// TIA Portal V15.1 export
// export: Created 2024-06-21T08:40:59.2288324Z, ExportSetting WithDefaults, DisplayName Totally Integrated Automation Portal, DisplayVersion V15.1 Update 5, DisplayName TIA Portal Openness, DisplayVersion V15.1 Update 5, DisplayName SINAMICS Startdrive Advanced, DisplayVersion V15.1, DisplayName G130, G150, S120, S150, SINAMICS MV, S210, DisplayVersion V15.1, DisplayName G110M, G120, G120C, G120D, G120P, DisplayVersion V15.1, DisplayName STEP 7 Professional, DisplayVersion V15.1 Update 5, DisplayName STEP 7 Safety, DisplayVersion V15.1, DisplayName WinCC Professional, DisplayVersion V15.1 Update 5, DisplayName SIMATIC Visualization Architect, DisplayVersion V15.1
FUNCTION_BLOCK "LVDComSubSystemS7-1500"   // FB2215, FBD
TITLE = VDComSubSystemS7-1500
{ S7_Optimized_Access := 'FALSE' }
AUTHOR : VCC
FAMILY : Communic
VERSION : 0.1
// =============================================================================
// This Module Extract Data From VDCom Send/Recv
// =============================================================================
// stored: AutoNumber false, IsIECCheckEnabled false, SetENOAutomatically False, UDAEnableTagReadback false
   VAR_INPUT
      I_CommunicationReset { ExternalAccessible := 'False'; ExternalVisible := 'False'; ExternalWritable := 'False'} : Bool;   // Reset communication by Application
      I_SendRequest { ExternalAccessible := 'False'; ExternalVisible := 'False'; ExternalWritable := 'False'} : Bool;   // Send Command by Application
      I_ResetNewData { ExternalAccessible := 'False'; ExternalVisible := 'False'; ExternalWritable := 'False'} : Bool;   // Trigger by Application to Reset output "NewData"
      I_MasterNewMessage { ExternalAccessible := 'False'; ExternalVisible := 'False'; ExternalWritable := 'False'} : Bool;   // Signal from MasterBlock to indicate new message.
      I_MasterSendFinished { ExternalAccessible := 'False'; ExternalVisible := 'False'; ExternalWritable := 'False'} : Bool;   // Acknowledge from MasterBlock that Send command has been performed
      I_VDCommRecvDB { ExternalAccessible := 'False'; ExternalVisible := 'False'; ExternalWritable := 'False'} : DB_ANY;   // VD communication system receive DB; Not to be used by Application
      I_VDCommSendDB { ExternalAccessible := 'False'; ExternalVisible := 'False'; ExternalWritable := 'False'} : DB_ANY;   // VD communication system send DB; Not to be used by Application
      C_LocalRecvDB { ExternalAccessible := 'False'; ExternalVisible := 'False'; ExternalWritable := 'False'} : DB_ANY;   // Local DB For Recv Data Used By The Application
      C_LocalSendDB { ExternalAccessible := 'False'; ExternalVisible := 'False'; ExternalWritable := 'False'} : DB_ANY;   // Local DB For Send Data Used By The Application
      C_MessType { ExternalAccessible := 'False'; ExternalVisible := 'False'; ExternalWritable := 'False'} : Int := 10;   // Identify Message
      C_SubSystem { ExternalAccessible := 'False'; ExternalVisible := 'False'; ExternalWritable := 'False'} : Int;   // Identify Subsystem
      C_SendMessLen { ExternalAccessible := 'False'; ExternalVisible := 'False'; ExternalWritable := 'False'} : Word;   // Number to identify the Length of the message
   END_VAR
   VAR_OUTPUT
      O_SendFinished { ExternalAccessible := 'False'; ExternalVisible := 'False'; ExternalWritable := 'False'} : Bool;   // Sending of Data is done; to Application
      O_NewData { ExternalAccessible := 'False'; ExternalVisible := 'False'; ExternalWritable := 'False'} : Bool;   // New data is available from SubSystem to Application
   END_VAR
   VAR_IN_OUT
      IO_MasterSendReq { ExternalAccessible := 'False'; ExternalVisible := 'False'; ExternalWritable := 'False'} : Bool;   // Request from the SubBlock to the MasterBlock to Send data
      IO_MasterAckReq { ExternalAccessible := 'False'; ExternalVisible := 'False'; ExternalWritable := 'False'} : Bool;   // Acknowledge to Master upon MessageType- and SubSystem Match
      IO_SubSystemDBNr { ExternalAccessible := 'False'; ExternalVisible := 'False'; ExternalWritable := 'False'} : Int;   // VD Communication Send DB number, Set by SubSystem
      IO_VDCommSendDB { ExternalAccessible := 'False'; ExternalVisible := 'False'; ExternalWritable := 'False'} : DB_ANY;   // VD Communication send DB
   END_VAR
   VAR DB_SPECIFIC
      ThisModuleActiveSend { ExternalAccessible := 'False'; ExternalVisible := 'False'; ExternalWritable := 'False'} : Bool;   // This module active for sending
      ThisModuleActiveRead { ExternalAccessible := 'False'; ExternalVisible := 'False'; ExternalWritable := 'False'} : Bool;   // This module active for Reading / acknowledge
      NewDataPulse { ExternalAccessible := 'False'; ExternalVisible := 'False'; ExternalWritable := 'False'} : Bool;   // Bit to create pulse on NewData
      NewData { ExternalAccessible := 'False'; ExternalVisible := 'False'; ExternalWritable := 'False'} : Bool;   // New Data
      NewDataAvailable { ExternalAccessible := 'False'; ExternalVisible := 'False'; ExternalWritable := 'False'} : Bool;   // New Data Available
      NewDataAvailablePulse { ExternalAccessible := 'False'; ExternalVisible := 'False'; ExternalWritable := 'False'} : Bool;   // New Data Available Pulse
      _RestartSend { ExternalAccessible := 'False'; ExternalVisible := 'False'; ExternalWritable := 'False'; S7_SetPoint := 'True'} : IEC_TIMER;
   END_VAR
   VAR_TEMP
      PtrRECV : Any;   // Pointer to the system receive DB
      PtrARECV : Any;   // Pointer to the Application receive DB
      RecvMessType : Int;   // Message type of the received data
      RecvSubSyst : Int;   // Subsystem target number
      RcvLength : Int;   // Length of received data
      RecvDBNbr : Int;   // Receive system DB Number
      SendDBNbr : Int;   // Send system DB Number
      LocalRecvDBNbr : Int;   // Receive DB Number Local by Application
      LocalSendDBNbr : Int;   // Send DB Number Local by Application
   END_VAR
   VAR_TEMP   // added for the SCL form of the ladder/FBD networks
      _w1 : Bool;
      _w2 : Bool;
   END_VAR
BEGIN

NETWORK
TITLE = **** 1 - Inputs **** Load DB
// Load DB numbers to local variables from the Receive and Send DB from - VD Master - VD Subsystem
// Read DB Number Recv
      OPN   #I_VDCommRecvDB;
      L     DBNO;
      T     #RecvDBNbr;

// Read DB Number Send
      OPN   #I_VDCommSendDB;
      L     DBNO;
      T     #SendDBNbr;

// DB Number from VD Sub system
      OPN   #C_LocalRecvDB;
      L     DBNO;
      T     #LocalRecvDBNbr;

// Read DB Number Send
      OPN   #C_LocalSendDB;
      L     DBNO;
      T     #LocalSendDBNbr;

REGION Network 2: **** 3.1 - Communication - Other Systems **** Reset Communications
   // Reset Communications
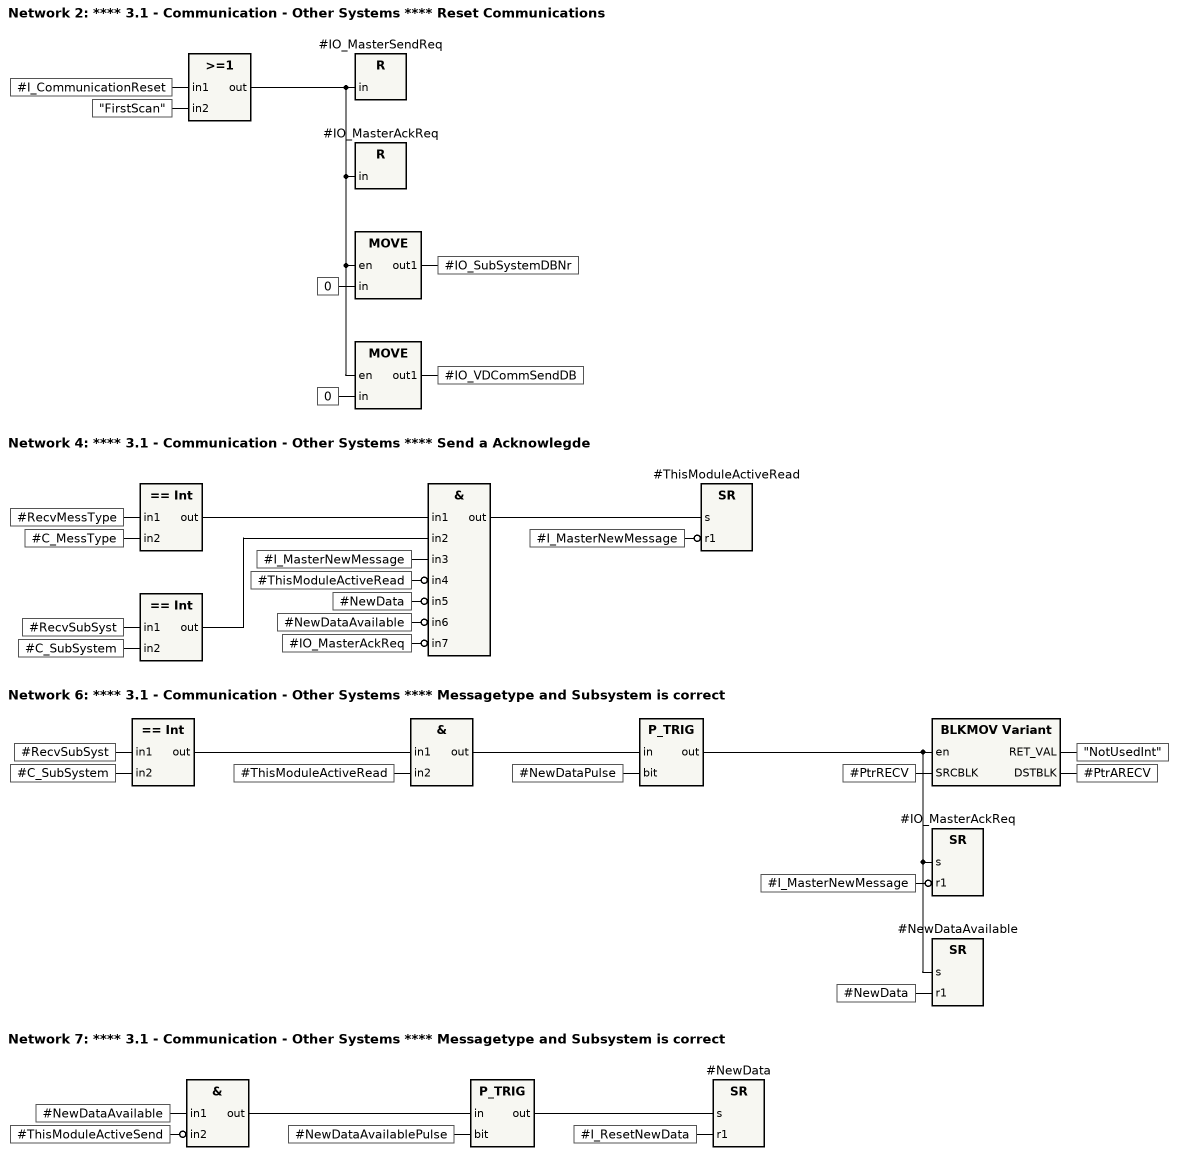
   IF #I_CommunicationReset OR "FirstScan" THEN
       #IO_MasterSendReq := FALSE;
       #IO_MasterAckReq := FALSE;
       #IO_SubSystemDBNr := 0;
       #IO_VDCommSendDB := 0;
   END_IF;
END_REGION

NETWORK
TITLE = **** 3.1 - Communication - Other Systems **** Header Information
// Copy Header information to local variables  Copy MessageType to local variable
      A     #ThisModuleActiveRead;
      JC    TMAR;
//OPN DB [ #RecvDBNbr] APa S7-1500
      OPN   #I_VDCommRecvDB;
      L     %DBW4;
      T     #RecvMessType;
//Copy SubSystemNbr to local variable
      L     %DBW6;
      T     #RecvSubSyst;
//Copy Lenth to local variable
      L     %DBW2;
      T     #RcvLength;
TMAR: NOP   0;

REGION Network 4: **** 3.1 - Communication - Other Systems **** Send a Acknowlegde
   // Send a Acknowlegde Request if Messagetype and Subsystem is correct
   IF (#RecvMessType = #C_MessType) AND (#RecvSubSyst = #C_SubSystem) AND #I_MasterNewMessage AND NOT #ThisModuleActiveRead AND NOT #NewData AND NOT #NewDataAvailable AND NOT #IO_MasterAckReq THEN
       #ThisModuleActiveRead := TRUE;   // SR flip-flop
   END_IF;
   IF NOT #I_MasterNewMessage THEN #ThisModuleActiveRead := FALSE; END_IF;
END_REGION

NETWORK
TITLE = **** 3.1 - Communication - Other Systems **** Configure DB
// Configure DB pointers
// APa Cleaning Warnings
      LAR1  P##PtrRECV;
      L     16#1002;
      T     LW [AR1, P#0.0];
      L     #RcvLength;
      T     LW [AR1, P#2.0];
      L     #RecvDBNbr;
      T     LW [AR1, P#4.0];
      L     0;
      SLD   3;
      OD    16#8400_0000;
      T     LD [AR1, P#6.0];

      LAR1  P##PtrARECV;
      L     16#1002;
      T     LW [AR1, P#0.0];
      L     #RcvLength;
      T     LW [AR1, P#2.0];
      L     #LocalRecvDBNbr;
      T     LW [AR1, P#4.0];
      L     0;
      SLD   3;
      OD    16#8400_0000;
      T     LD [AR1, P#6.0];
//      L     16#10                // S7  S7
//      T     %LB0
//      T     %LB10
//      L     16#02                // Data type to copy B#16#2 = Bytes
//      T     %LB1
//      T     %LB11
//      L     #RcvLength           //Length receiving data
//      T     %LW2
//      T     %LW12
//      L     #RecvDBNbr           // Receive DB Number
//      T     %LW4
//      L     #LocalRecvDBNbr      // Local Receive DB Number
//      T     %LW14
//      L     L#0                  //Offset in DB
//      SLD   3                    // Convert to pointer
//      T     %LD6
//      T     %LD16
//      L     16#84                // Memory area DB Memory area DB
//      T     %LB6
//      T     %LB16


REGION Network 6: **** 3.1 - Communication - Other Systems **** Messagetype and Subsystem is correct
   // New Data-flag if Messagetype and Subsystem is correct
   #_w1 := (#RecvSubSyst = #C_SubSystem) AND #ThisModuleActiveRead;
   #_w2 := #_w1 AND NOT #NewDataPulse;   // rising edge
   #NewDataPulse := #_w1;
   IF #_w2 THEN
       "NotUsedInt" := BLKMOV(SRCBLK := #PtrRECV, DSTBLK => #PtrARECV);
       #IO_MasterAckReq := TRUE;   // SR flip-flop
   END_IF;
   IF NOT #I_MasterNewMessage THEN #IO_MasterAckReq := FALSE; END_IF;
   IF #_w2 THEN
       #NewDataAvailable := TRUE;   // SR flip-flop
   END_IF;
   IF #NewData THEN #NewDataAvailable := FALSE; END_IF;
END_REGION

REGION Network 7: **** 3.1 - Communication - Other Systems **** Messagetype and Subsystem is correct
   // New Data-flag if Messagetype and Subsystem is correct
   #_w1 := #NewDataAvailable AND NOT #ThisModuleActiveSend;
   #_w2 := #_w1 AND NOT #NewDataAvailablePulse;   // rising edge
   #NewDataAvailablePulse := #_w1;
   IF #_w2 THEN
       #NewData := TRUE;   // SR flip-flop
   END_IF;
   IF #I_ResetNewData THEN #NewData := FALSE; END_IF;
END_REGION

NETWORK
TITLE = **** 3.1 - Communication - Other Systems **** Configure Header
// Configure Header for send data
//      OPN DB [ #LocalSendDBNbr] APa S7-1500
      OPN   #C_LocalSendDB;
      L     16#01;  //VD Version
      T     %DBB0;

      L     16#00;  //spare byte
      T     %DBB1;

//
      L     #C_SendMessLen;
      L     0;
      ==I;
      JC    Len1;
      L     #C_SendMessLen;
      JU    Len2;
Len1: L     DBLG;
Len2: T     %DBW2;

      L     #C_MessType;
      T     %DBW4;

      L     #C_SubSystem;
      T     %DBW6;


REGION Network 9: **** 3.1 - Communication - Other Systems **** This module is Active for Sending
   // This Module Active For Sending
   // - Check if no Request active (IO_MasterSendReq)
   // - Check if No DB Selected
   // - Check if Master does not send finished
   // - Send data Request from Application
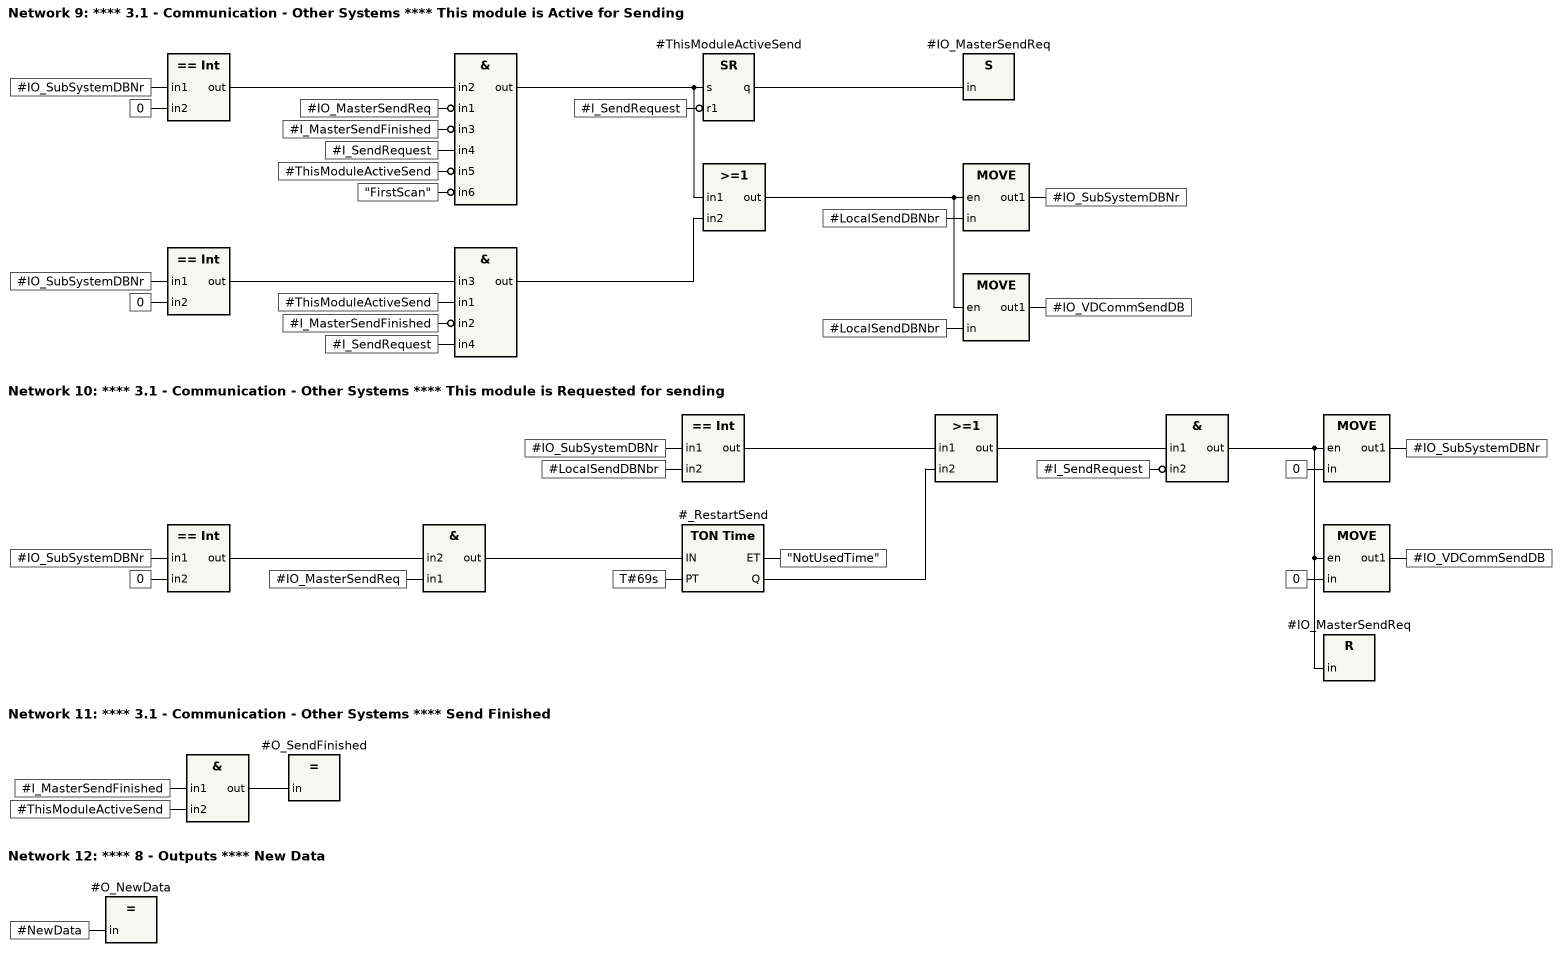
   #_w1 := (#IO_SubSystemDBNr = 0) AND NOT #IO_MasterSendReq AND NOT #I_MasterSendFinished AND #I_SendRequest AND NOT #ThisModuleActiveSend AND NOT "FirstScan";
   IF #_w1 THEN
       #ThisModuleActiveSend := TRUE;   // SR flip-flop
   END_IF;
   IF NOT #I_SendRequest THEN #ThisModuleActiveSend := FALSE; END_IF;
   IF #ThisModuleActiveSend THEN #IO_MasterSendReq := TRUE; END_IF;
   #_w2 := #_w1 OR ((#IO_SubSystemDBNr = 0) AND #ThisModuleActiveSend AND NOT #I_MasterSendFinished AND #I_SendRequest);
   IF #_w2 THEN
       #IO_SubSystemDBNr := #LocalSendDBNbr;
       #IO_VDCommSendDB := #LocalSendDBNbr;
   END_IF;
END_REGION

REGION Network 10: **** 3.1 - Communication - Other Systems **** This module is Requested for sending
   // This module is Requested for sending
   #_RestartSend.TON(IN := (#IO_SubSystemDBNr = 0) AND #IO_MasterSendReq, PT := T#69s, ET => "NotUsedTime");
   #_w1 := ((#IO_SubSystemDBNr = #LocalSendDBNbr) OR #_RestartSend.Q) AND NOT #I_SendRequest;
   IF #_w1 THEN
       #IO_SubSystemDBNr := 0;
       #IO_VDCommSendDB := 0;
       #IO_MasterSendReq := FALSE;
   END_IF;
END_REGION

REGION Network 11: **** 3.1 - Communication - Other Systems **** Send Finished
   // Send Finished
   #O_SendFinished := #I_MasterSendFinished AND #ThisModuleActiveSend;
END_REGION

REGION Network 12: **** 8 - Outputs **** New Data
   // New Data
   #O_NewData := #NewData;
END_REGION
END_FUNCTION_BLOCK
